TYPE DUT_HMI_Out_Resource :
STRUCT
	Origin : DUT_OutInfoOrigin;
END_STRUCT
END_TYPE

(* stored: Version 1.1.0.1, ProductVersion 3.1.4024.13
   DUT DUT_HMI_Out_Resource: Id {d33f3e2c-1726-44f5-842b-e4fe9eaf20d1} *)
